FUNCTION_BLOCK FB_FootPedal
VAR_INPUT
	PedalPressed1			:BOOL;	
	PedalPressed2			:BOOL;
	PedalPressed3			:BOOL;
	debounce_time			:LREAL;//ms The amount of time that the foot pedal does not register another click.	
END_VAR
VAR_OUTPUT
	error_code					:INT;	//	
	state					:INT;	//	
	pressed					:INT;//‘none’, ‘pedal1’, ‘pedal2’, ‘pedal3’	
	Error					:BOOL;
END_VAR
VAR
	ton1:Tc2_Standard.TON;
	step:INT;
	TRIG1:Tc2_Standard.R_TRIG;
END_VAR
VAR_IN_OUT
	Reset					:BOOL;
END_VAR

CASE step OF
0:
	state:=FootPedalStateEnum.ready;
	error_code:=FootPedalErrorEnum.no_error;
	pressed:=0;
	ton1(IN:=FALSE);
	Reset:=FALSE;
	
	IF PedalPressed1 THEN 
		step:=10;
	ELSIF PedalPressed2 THEN 
		step:=20;
	ELSIF PedalPressed3 THEN 
		step:=30;
	END_IF
	
10:	
	IF PedalPressed1 THEN 
		pressed:=1;
	ELSE 
		pressed:=0;
		step:=50;
	END_IF
	
20:	
	IF PedalPressed2 THEN 
		pressed:=2;
	ELSE 
		pressed:=0;
		step:=50;
	END_IF

30:	
	IF PedalPressed3 THEN 
		pressed:=3;
	ELSE 
		pressed:=0;
		step:=50;
	END_IF

50://缓冲
	ton1(IN:=TRUE , PT:=LREAL_TO_TIME(debounce_time) , Q=> , ET=> );
	IF ton1.Q THEN 
		step:=0;
	END_IF
100://error
	state:=FootPedalStateEnum.error;
	pressed:=0;
	error:=TRUE;
	IF Reset OR GVL.Reset THEN 
		Reset:=FALSE;
		error:=FALSE;
		step:=0;
	END_IF
END_CASE

IF Reset OR GVL.Reset THEN 
	Reset:=FALSE;
	error:=FALSE;
	step:=0;
END_IF


TRIG1(CLK:=GVL.Emstop_Button , Q=> ); 
	IF TRIG1.Q THEN 
		error_code:=FootPedalErrorEnum.emergency_error;
		step:=100;
	END_IF

END_FUNCTION_BLOCK

(* stored: Version 1.1.0.1, ProductVersion 3.1.4024.11
   POU FB_FootPedal: Id {17f0628c-709c-4286-9d98-7c29f7d841f8}, SpecialFunc None *)
